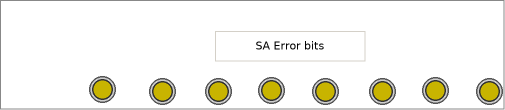
VISUALIZATION Visualization  // 505x110
    Lamp1 (310,73 31x37), variable: MAIN.err_ff, style: Lamp-Lamp1-Yellow
    Lamp1 (256,72 31x37), variable: MAIN.err_f_step, style: Lamp-Lamp1-Yellow
    Lamp1 (203,73 31x37), variable: MAIN.err_f_minmax, style: Lamp-Lamp1-Yellow
    Lamp1 (147,73 31x37), variable: MAIN.err_dongle, style: Lamp-Lamp1-Yellow
    Lamp1 (87,71 31x37), variable: MAIN.err_cal, style: Lamp-Lamp1-Yellow
    Lamp1 (474,73 31x37), variable: MAIN.err_soc, style: Lamp-Lamp1-Yellow
    Lamp1 (420,72 31x37), variable: MAIN.err_mhb, style: Lamp-Lamp1-Yellow
    Lamp1 (367,73 31x37), variable: MAIN.err_locid, style: Lamp-Lamp1-Yellow
    Textfield (215,31 150x30), "SA Error bits"
END_VISUALIZATION

(* stored: Version 1.1.0.1, ProductVersion 3.1.4024.9
   Visu Visualization: Id {68795125-2f9d-4e6f-8718-d56ba967191b} *)
